PROGRAM MAIN
VAR
	fbTon: Tc2_Standard.TON;
END_VAR

fbTon(IN:=NOT fbTon.Q , PT:=T#1S , Q=> , ET=> );

IF fbTon.Q THEN
	// Update bool
	GVL_Test.bTestRead := NOT GVL_Test.bTestRead;
	// Update real
	IF GVL_Test.fTestRead < 10.0 THEN
		GVL_Test.fTestRead := GVL_Test.fTestRead + 0.5;
	ELSE
		GVL_Test.fTestRead := -10.0;
	END_IF
END_IF

END_PROGRAM

(* stored: Version 1.1.0.1, ProductVersion 3.1.4024.6
   POU MAIN: Id {9226b76d-0684-4b68-b80b-43dc2364f929}, SpecialFunc None *)
